PROGRAM MAIN
VAR
	{region 'Settings'}
		DPAD					: FB_BA_CarelessDPAD:=(
									aIdentifier:=[
										(* Level 1 *)	(eNodeType:=E_BA_NodeType.eBuilding,	nIndexDigits:=2),
										(* Level 2 *)	(eNodeType:=E_BA_NodeType.eTrade,		nIndexDigits:=0),
										(* Level 3 *)	(eNodeType:=E_BA_NodeType.ePlant,		nIndexDigits:=2,			sSeparator_ObjectName:='~~~',		sSeparator_Description:=' --- '),
										(* Level 4 *)	(eNodeType:=E_BA_NodeType.eAggregate,	nIndexDigits:=2,			sSeparator_ObjectName:='++'),
										(* Level 5 *)	(eNodeType:=E_BA_NodeType.eFunction,	nIndexDigits:=3)
								]);
	{endregion}
		 
	Smpl						: FB_BA_View			:= (									sDescription:='Samples');
	{region 'Demonstration'}
		Demo					: FB_BA_View			:= (iParent:=Smpl,						sDescription:='Demonstration');
			Obj					: FB_BA_View			:= (iParent:=Demo,						sDescription:='Objects');
				General			: FB_Obj_General		:= (iParent:=Obj,						sDescription:='General objects');
				Misc			: FB_Obj_Misc			:= (iParent:=Obj,						sDescription:='Miscellaneous objects');
				Seq				: FB_Obj_Sequence		:= (iParent:=Obj,						sDescription:='Sequences');
				UdObj			: FB_Obj_UserDefined	:= (iParent:=Obj,						sDescription:='User defined objects');
				AddParam		: FB_Obj_AddParam		:= (iParent:=Obj,						sDescription:='Additional parameters');
					 
			Ref					: FB_BA_View			:= (iParent:=Demo,						sDescription:='Reference');
				Collect			: FB_Ref_Collectors		:= (iParent:=Ref,						sDescription:='Collectors');
				Groups			: FB_Ref_Groups			:= (iParent:=Ref,						sDescription:='Groups');
				PubSubLc		: FB_Ref_PubSub_Local	:= (iParent:=Ref,						sDescription:='Publisher and subscriber (Local)');
				PubSubRm		: FB_Ref_PubSub_Remote	:= (iParent:=Ref,						sDescription:='Publisher and subscriber (Remote)');
					 
			Evt					: FB_BA_View			:= (iParent:=Demo,						sDescription:='Event');
				EvtCls			: FB_Evt_EventClasses	:= (iParent:=Evt,						sDescription:='Event classes');
				Events			: FB_Evt_Events			:= (iParent:=Evt,						sDescription:='Events');
				Ack				: FB_Evt_Ack			:= (iParent:=Evt,						sDescription:='Acknowledgement');
				MiscEvt			: FB_Evt_Misc			:= (iParent:=Evt,						sDescription:='Miscellaneous');
					 
			Strct				: FB_BA_View			:= (iParent:=Demo,						sDescription:='Structure');
				Nested			: FB_Struct_Nested		:= (iParent:=Strct,						sDescription:='Nested objects');
					 
			Plt					: FB_BA_View			:= (iParent:=Demo,						sDescription:='Plant');
				PltCtrl1		: FB_Plt_Init1			:= (iParent:=Plt,						sDescription:='Plant control initialization 1');
				PltCtrl2		: FB_Plt_Init2			:= (iParent:=Plt,						sDescription:='Plant control initialization 2');
				PltCtrl3		: FB_Plt_Init3			:= (iParent:=Plt,						sDescription:='Plant control initialization 3');
					 
			Spl					: FB_BA_View			:= (iParent:=Demo,						sDescription:='Supplement specific');
				BACnet_RcpList	: FB_BACnet_RcpList		:= (iParent:=Spl,						sDescription:='Recipient list (BACnet)');
				BACnet_Flags	: FB_BACnet_StatusFlags;	 
			Other				: FB_BA_View			:= (iParent:=Demo,						sDescription:='Other');
				MscOth			: FB_Misc				:= (iParent:=Other,						sDescription:='Miscellaneous');
	{endregion}
	{region 'Templates'}
		Tmpl					: FB_BA_View			:= (iParent:=Smpl,						sDescription:='Templates');
			Gen					: FB_BA_View			:= (iParent:=Tmpl,						sDescription:='General');
				Bld01			: FB_BA_Bld01			:= (iParent:=Gen,						sDescription:='Building information');
				EvtCls01		: FB_BA_EC01			:= (iParent:=Gen,						sDescription:='Event Classes');
	{endregion}		
END_VAR
VAR		
	nCounter					: UDINT					:= 0;	
END_VAR

nCounter:=(nCounter+1);

Smpl();

// Demonstration:
Demo();

Obj();
General();
Misc();
Seq();
UdObj();
AddParam();

Ref();
Collect();
Groups();
PubSubLc();
PubSubRm();

Evt();
EvtCls();
Events();
Ack();
MiscEvt();

Strct();
Nested();

Plt();
PltCtrl1();
PltCtrl2();
PltCtrl3();

Spl();
BACnet_RcpList();
BACnet_Flags();

Other();
MscOth();

// Templates:
Tmpl();

Gen();
Bld01();
EvtCls01();

// Optional extensions:
MAIN_OPTEXT();

END_PROGRAM

(* stored: Version 1.1.0.1, ProductVersion 3.1.4024.12
   POU MAIN: Id {7c15d84c-41a4-421d-9b24-c13041281be0}, SpecialFunc None *)
